# EPICS SNL sequencer program: mm4006App/src/mm4006.stt
//###############################################
//# ###										### #
//# ### Epics SNL Routines for				### #
//# ### Status Motor Device			### #
//# ###										### #
//# ### author: D. Hampai - M. Montis		### #
//# ###										### #
//# ### Ref 2.0; 2026-08-02					### #
//###############################################
//#
//
program sncmm4006
//
%{
#include <math.h>
#include <stdlib.h>
#include <unistd.h>
#include <time.h>
#include <sys/stat.h>
#include <errno.h>
#include <epicsThread.h>
#include "motor_status.h"
#include "res_utils.h"

// Dichiarazione globale della variabile MotorStatus
MotorStatus g_motor_status;
char g_motor_status_char;
TotalStatus g_motor_status_opt;
char g_motor_status_opt_char;
}%
//
option +r;
/*	PV/CA Variables
Num	Name			type		Associated

1	mres			float		{motor}_{card}_{axis}:mres
2	polarity		int		{motor}_{card}_{axis}:polarity
3	status_mode		int		{motor}_{card}_{axis}:status_mode
4	ask_request		int		{motor}_{card}_{axis}:ask_request
5	check_err		stringin	{motor}_{card}_{axis}:err
6	ms_status		stringin	{motor}_{card}_{axis}:ms_status
7	ms_status_opt		stringin	{motor}_{card}_{axis}:ms_status_opt
8	motor_status		int		{motor}_{card}_{axis}:motor_status
9	lim_pos			int		{motor}_{card}_{axis}:limit_right
10	lim_neg			int		{motor}_{card}_{axis}:limit_left
11	mot_moving		int		{motor}_{card}_{axis}:moving
12	reqpos			int		{motor}_{card}_{axis}:reqpos
13	atc_pos			float		{motor}_{card}_{axis}:act_pos
14	pos			float		{motor}_{card}_{axis}:pos
15	reqvel			int		{motor}_{card}_{axis}:reqvel
16	act_vel			float		{motor}_{card}_{axis}:act_vel
17	real_vel		float		{motor}_{card}_{axis}:real_vel
*/

/*	Local Variables
int status_mode;
*/
// PV/CA
float mres; assign mres to "{motor}_{card}_{axis}:mres"; monitor mres;
int polarity; assign polarity to "{motor}_{card}_{axis}:polarity"; monitor polarity;
int status_mode; assign status_mode to "{motor}_{card}_{axis}:status_mode"; monitor status_mode;
int ask_request; assign ask_request to "{motor}_{card}_{axis}:ask_request"; monitor ask_request;
string check_err; assign check_err to "{motor}_{card}_{axis}:err"; monitor check_err;
string ms_status; assign ms_status to "{motor}_{card}_{axis}:ms_status"; monitor ms_status;
string ms_status_opt; assign ms_status_opt to "{motor}_{card}_{axis}:ms_status_opt"; monitor ms_status_opt;
int  motor_status; assign motor_status to "{motor}_{card}_{axis}:motor_status"; monitor motor_status;
int lim_pos; assign lim_pos to "{motor}_{card}_{axis}:limit_right"; monitor lim_pos;
int lim_neg; assign lim_neg to "{motor}_{card}_{axis}:limit_left"; monitor lim_neg;
int mot_moving; assign mot_moving to "{motor}_{card}_{axis}:moving"; monitor mot_moving;
int reqpos; assign reqpos to "{motor}_{card}_{axis}:reqpos"; monitor reqpos;
float act_pos; assign act_pos to "{motor}_{card}_{axis}:act_pos"; monitor act_pos;
float pos; assign pos to "{motor}_{card}_{axis}:pos"; monitor pos;
int reqvel; assign reqvel to "{motor}_{card}_{axis}:reqvel"; monitor reqvel;
float act_vel; assign act_vel to "{motor}_{card}_{axis}:act_vel"; monitor act_vel;
float real_vel; assign real_vel to "{motor}_{card}_{axis}:real_vel"; monitor real_vel;

// PV/CA .PROC
int ms_status_proc; assign ms_status_proc to "{motor}_{card}_{axis}:ms_status.PROC";
int ms_status_opt_proc; assign ms_status_opt_proc to "{motor}_{card}_{axis}:ms_status_opt.PROC";

//Local Variables
// int status_mode;
string lc_motor;
string lc_card;
string lc_axis;
string actual_motor;
char motor_status_char;
char motor_status_opt_char;
string motor_name;
int ismoving;
float get_pol;
//
//
ss motor_snl {
	state init {
		when () {
			strcpy(lc_motor,macValueGet("motor"));
			strcpy(lc_card,macValueGet("card"));
			strcpy(lc_axis,macValueGet("axis"));
			status_mode = 0;
			pvPut(status_mode, SYNC);
			printf("Init done\n");
			pvGet(mres,SYNC);
			pvGet(polarity,SYNC);
			get_pol = 1;
		} state idle
	}
//
	state idle {
		when(status_mode==1) {
			printf("motor %s, card %s, axis %s, status_mode %d\n", lc_motor, lc_card, lc_axis, status_mode);
//			status_mode=0;
//			pvPut(status_mode,SYNC);
			epicsThreadSleep(1.0);
		} state check_err
		when(reqpos==1) {
			printf("Request Position\n");
			status_mode=3;
			pvPut(status_mode,SYNC);
		} state check_err
		when(reqvel==1) {
			printf("Request Velocity\n");
			status_mode=4;
			pvPut(status_mode,SYNC);
		} state check_err
		when() {
//			serve solo per debug... poi da togliere
//			printf("IOC%s_%s waiting for check", lc_card, lc_axis);
			epicsThreadSleep(1.0);
		} state idle
	}
//
	state check_status {
		when () {
//			MotorStatus ms;
			ms_status_proc = 1;
			pvPut(ms_status_proc, SYNC);
			epicsThreadSleep(0.1);
//
	 		pvGet(ms_status, SYNC);
			motor_status_char = ms_status[0];
//			motor_status_char = (char)ms_status;
//
			parse_motor_status(motor_status_char, &g_motor_status);
//
			/* Usa i singoli campi */
			if (!g_motor_status.power_on) {
				printf("ERRORE: motore spento!\n");
			}
			if (g_motor_status.limit_right || g_motor_status.limit_left) {
				printf("ATTENZIONE: limite scattato!\n");
			}
			if (g_motor_status.in_motion) {
				printf("Motore in movimento (%s)\n", g_motor_status.dir_positive ? "+" : "-");
			}
			printf("%d,%d,%d,%d\n", g_motor_status.power_on, g_motor_status.limit_right, g_motor_status.limit_left, g_motor_status.in_motion);
//
			motor_status = g_motor_status.power_on;
			pvPut(motor_status,SYNC);
			lim_pos = g_motor_status.limit_right;
			pvPut(lim_pos,SYNC);
			lim_neg = g_motor_status.limit_left;
			pvPut(lim_neg,SYNC);
			/* Oppure debug rapido */
			sprintf(motor_name,"Motor%s", lc_axis);
			print_motor_status(motor_name, motor_status_char);
			status_mode=2;
			pvPut(status_mode,SYNC);
//			print_motor_status("Motor1", motor_status_char);
		} state check_err
	}
// motor_status_opt_char
	state check_status_opt {
		when() {
			ms_status_opt_proc = 1;
			pvPut(ms_status_opt_proc,SYNC);
			epicsThreadSleep(0.1);
//
			pvGet(ms_status_opt,SYNC);
			motor_status_opt_char = ms_status_opt[0];
//
//	Da Togliere... solo come prova per debug
//
//			printf("DEBUG TS raw string: '%s' primo char: 0x%02X (%d)\n", ms_status_opt,
//				(unsigned char)ms_status_opt[0],
//				(unsigned char)ms_status_opt[0]);
//			g_motor_status_opt_char = (char)ms_status_opt;
//
			parse_total_status(motor_status_opt_char, &g_motor_status_opt);
//
			if (lc_axis == 1) {
				mot_moving = g_motor_status_opt.axis1_moving;
			} else if (lc_axis == 2) {
				mot_moving = g_motor_status_opt.axis2_moving;
			} else if (lc_axis == 3) {
				mot_moving = g_motor_status_opt.axis3_moving;
			} else {
				mot_moving = g_motor_status_opt.axis4_moving;
			}
			pvPut(mot_moving,SYNC);
//
			/* Oppure debug rapido */
			print_total_status(motor_status_opt_char);
			status_mode=3;
			pvPut(status_mode,SYNC);
		} state check_err
	}
	state check_position {
		when() {
			pvPut(act_pos,SYNC);
			epicsThreadSleep(0.1);
//
			pvGet(act_pos,SYNC);
//			pos = mech_to_real(mres,act_pos,polarity);
			pos = mech_to_real(mres,act_pos,get_pol);
			printf("The position is %.3f\n", pos);
			pvPut(pos,SYNC);
			reqpos=0;
			pvPut(reqpos,SYNC);
//			status_mode=0;
			status_mode=4;
			pvPut(status_mode,SYNC);
		} state check_err
	}
	state check_velocity {
		when() {
			pvPut(act_vel,SYNC);
			epicsThreadSleep(0.1);
//
			pvGet(act_vel,SYNC);
			real_vel = mech_to_real(mres,act_vel,get_pol);
			printf("The velocity is %.3f\n", real_vel);
			pvPut(real_vel,SYNC);
			reqvel=0;
			pvPut(reqvel,SYNC);
			status_mode=0;
			pvPut(status_mode,SYNC);
		} state check_err
	}
	state check_err {
		when(status_mode==1) {
			printf("Check Error in State %d\n", status_mode);
			pvPut(check_err, SYNC);
		} state check_status
		when(status_mode==2) {
			printf("Check Error in State %d\n", status_mode);
			pvPut(check_err, SYNC);
		} state check_status_opt
		when(status_mode==3) {
			printf("Check Error in State %d\n", status_mode);
			pvPut(check_err, SYNC);
		} state check_position
		when(status_mode==4) {
			printf("Check Error in State %d\n", status_mode);
			pvPut(check_err, SYNC);
		} state check_velocity
		when() {
			printf("Check Error in State %d\n", status_mode);
			pvPut(check_err, SYNC);
		} state idle
	}
}
